// TIA Portal V17 export
// export: Created 2024-06-14T09:53:00.9899822Z, ExportSetting WithDefaults, DisplayName Totally Integrated Automation Portal, DisplayVersion V17, DisplayName TIA Portal Openness, DisplayVersion V17, DisplayName TIA Portal Version Control Interface, DisplayVersion V17, DisplayName Simotion SCOUT TIA, DisplayVersion 5.4.3.0, DisplayName SINAMICS Startdrive Advanced, DisplayVersion V17 SP1 Update 1, DisplayName SINAMICS Startdrive G110M, G120, G120C, G120D, G120P, G115D, DisplayVersion V17 SP1 Update 1, DisplayName SINAMICS Startdrive G130, G150, S120, S150, SINAMICS MV, S210, DisplayVersion V17 SP1 Update 1, DisplayName STEP 7 Professional, DisplayVersion V17, DisplayName STEP 7 Safety, DisplayVersion V17, DisplayName WinCC Professional, DisplayVersion V17
FUNCTION_BLOCK "keypad_logic"   // FB6, LAD
{ S7_Optimized_Access := 'TRUE' }
VERSION : 0.1
// stored: AutoNumber true, IsIECCheckEnabled false, IsRetainMemResEnabled false, MemoryReserve 100, SetENOAutomatically false, UDAEnableTagReadback false
   VAR_INPUT
      Num_0 : Bool;
      Num_1 : Bool;
      Num_2 : Bool;
      Num_3 : Bool;
      Num_4 : Bool;
      Num_5 : Bool;
      Num_6 : Bool;
      Num_7 : Bool;
      Num_8 : Bool;
      Num_9 : Bool;
      enter : Bool;
      clear : Bool;
   END_VAR
   VAR
      count_0 : CTU_INT;
   END_VAR
   VAR RETAIN
      Tens { S7_SetPoint := 'True'} : Int;
   END_VAR
   VAR
      ones : Int;
      decimal : Int;
      P_TRIG : Bool;
      MUL : Int;
      MUL_1 : Int;
      Tare_weight : Real;
      "count _reset" : Bool;
      Tare_Entry : Real;
      "screen count" : Int;
      screen_number : Int;
      screen_reset : Bool;
      MUL_2 : Int;
      count_1 : CTU_INT;
      count_cv_1 : Int;
      "BPCL COUNT" : Int;
      DOMESTIC : Bool;
      COMMERCIAL : Bool;
      MALALBAR_COUNT : Int;
   END_VAR
   VAR RETAIN
      SENSE_1 : Int;
      SENSE_2 : Int;
      SENSE_3 : Int;
      SENSE_4 : Int;
   END_VAR
   VAR
      "SENSI NG_TIME" : Int;
      sens_reset : Bool;
      "open screen" : Bool;
      DOMESTIC_1 : Bool;
      COMMERCIAL_1 : Bool;
      count_2 : CTU_INT;
   END_VAR
   VAR RETAIN
      password { S7_SetPoint := 'True'} : Int;
   END_VAR
   VAR
      password_1 : Int;
      password_2 : Int;
      password_3 : Int;
      password_4 : Int;
      password_5 : Int;
      mul_3 : Int;
      mul_4 : Int;
      mul_5 : Int;
      mul_6 : Int;
      password_reset : Bool;
      sens : Bool;
   END_VAR
   VAR_TEMP
      value_0 : Int;
      count_cv_0 : Int;
   END_VAR
   VAR_TEMP   // added for the SCL form of the ladder/FBD networks
      _w1 : Bool;
      _w2 : Bool;
      _w3 : Bool;
      _w4 : Bool;
      _w5 : Bool;
      _w6 : Bool;
   END_VAR
BEGIN

REGION Network 1
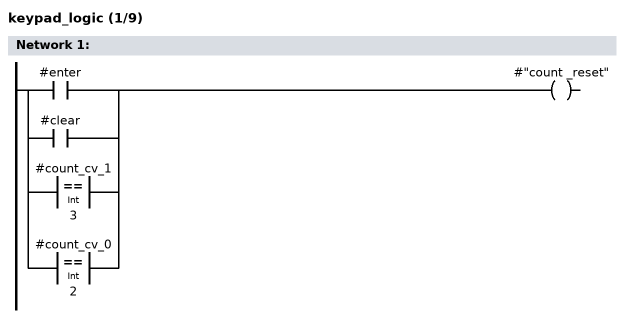
   RUNG wire#powerrail
      Contact( #enter )
      wire#w1
      Coil( #"count _reset" )
   END_RUNG
   RUNG wire#powerrail
      Contact( #clear )
   END_RUNG wire#w1
   RUNG wire#powerrail
      { S7_Templates := "SrcType := Int" } EQ_Contact(in1 := #count_cv_1, in2 := 3)
   END_RUNG wire#w1
   RUNG wire#powerrail
      { S7_Templates := "SrcType := Int" } EQ_Contact(in1 := #count_cv_0, in2 := 2)
   END_RUNG wire#w1
   // the same network as SCL:
   #"count _reset" := #enter OR #clear OR (#count_cv_1 = 3) OR (#count_cv_0 = 2);
END_REGION

REGION Network 2
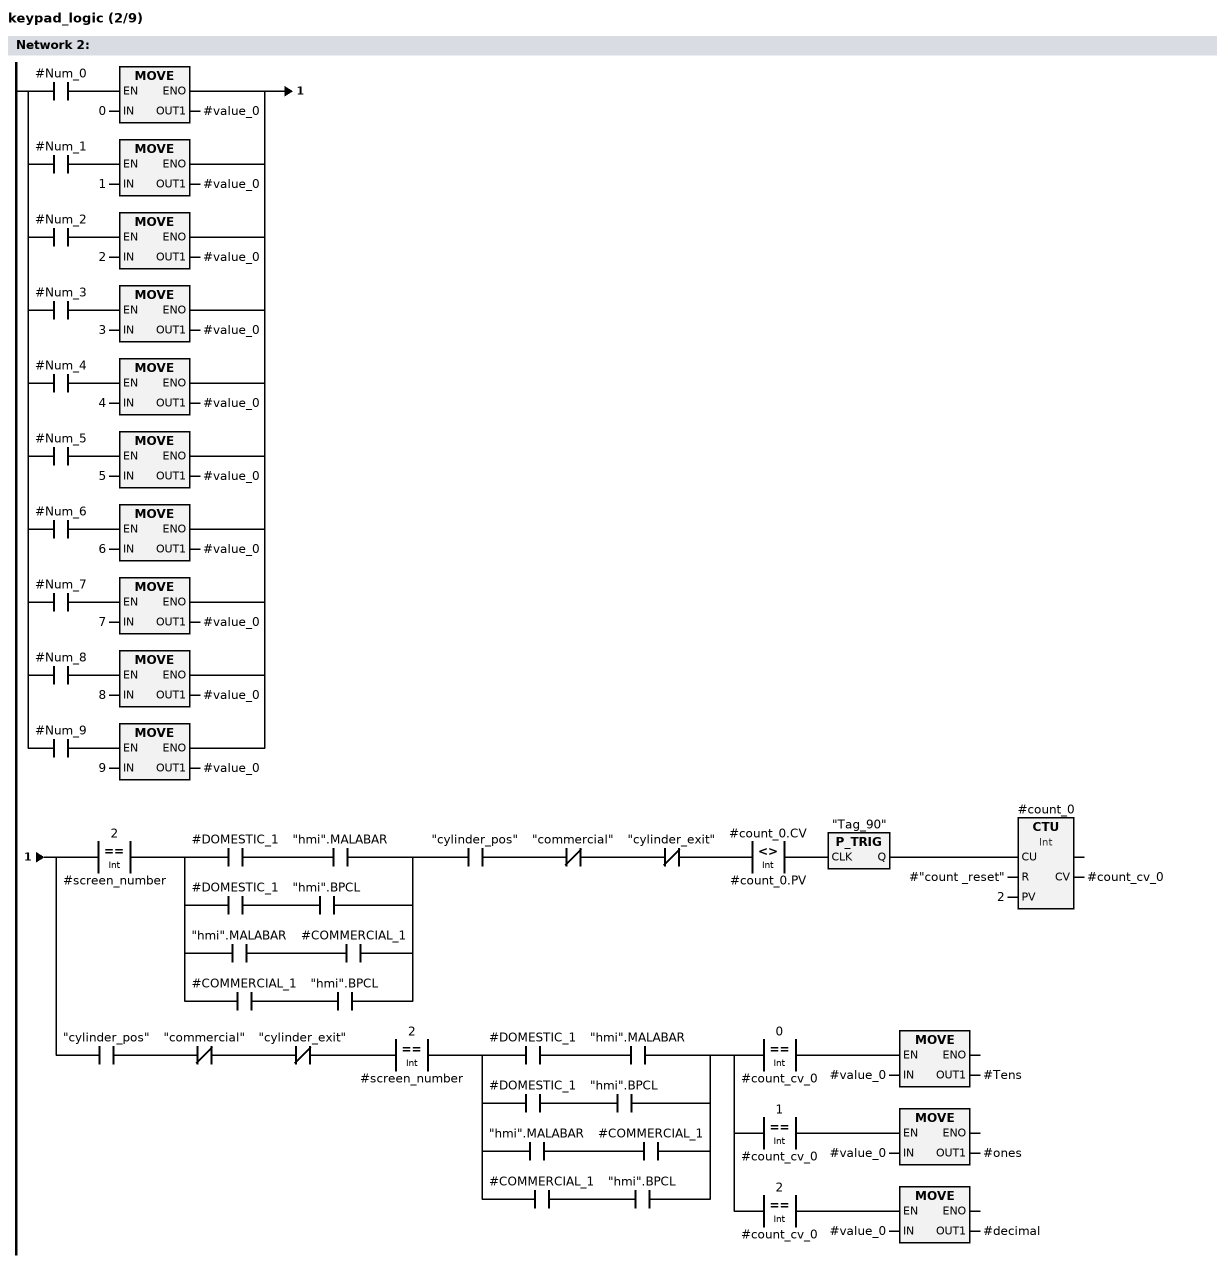
   RUNG wire#powerrail
      Contact( #Num_0 )
      Move(in := 0, out1 => #value_0)
      wire#w1
      { S7_Templates := "SrcType := Int" } EQ_Contact(in1 := 2, in2 := #screen_number)
      wire#w2
      Contact( #DOMESTIC_1 )
      Contact( "hmi".MALABAR )
      wire#w3
      Contact( "cylinder_pos" )
      I_Contact( "commercial" )
      I_Contact( "cylinder_exit" )
      { S7_Templates := "SrcType := Int" } NE_Contact(in1 := #count_0.CV, in2 := #count_0.PV)
      P_Trig( "Tag_90" )
      { S7_Templates := "value_type := Int" } #count_0.CTU(r := #"count _reset", pv := 2, cv => #count_cv_0)
   END_RUNG
   RUNG wire#powerrail
      Contact( #Num_1 )
      Move(in := 1, out1 => #value_0)
   END_RUNG wire#w1
   RUNG wire#powerrail
      Contact( #Num_2 )
      Move(in := 2, out1 => #value_0)
   END_RUNG wire#w1
   RUNG wire#powerrail
      Contact( #Num_3 )
      Move(in := 3, out1 => #value_0)
   END_RUNG wire#w1
   RUNG wire#powerrail
      Contact( #Num_4 )
      Move(in := 4, out1 => #value_0)
   END_RUNG wire#w1
   RUNG wire#powerrail
      Contact( #Num_5 )
      Move(in := 5, out1 => #value_0)
   END_RUNG wire#w1
   RUNG wire#powerrail
      Contact( #Num_6 )
      Move(in := 6, out1 => #value_0)
   END_RUNG wire#w1
   RUNG wire#powerrail
      Contact( #Num_7 )
      Move(in := 7, out1 => #value_0)
   END_RUNG wire#w1
   RUNG wire#powerrail
      Contact( #Num_8 )
      Move(in := 8, out1 => #value_0)
   END_RUNG wire#w1
   RUNG wire#powerrail
      Contact( #Num_9 )
      Move(in := 9, out1 => #value_0)
   END_RUNG wire#w1
   RUNG wire#w2
      Contact( #DOMESTIC_1 )
      Contact( "hmi".BPCL )
   END_RUNG wire#w3
   RUNG wire#w2
      Contact( "hmi".MALABAR )
      Contact( #COMMERCIAL_1 )
   END_RUNG wire#w3
   RUNG wire#w2
      Contact( #COMMERCIAL_1 )
      Contact( "hmi".BPCL )
   END_RUNG wire#w3
   RUNG wire#w1
      Contact( "cylinder_pos" )
      I_Contact( "commercial" )
      I_Contact( "cylinder_exit" )
      { S7_Templates := "SrcType := Int" } EQ_Contact(in1 := 2, in2 := #screen_number)
      wire#w4
      Contact( #DOMESTIC_1 )
      Contact( "hmi".MALABAR )
      wire#w5
      { S7_Templates := "SrcType := Int" } EQ_Contact(in1 := 0, in2 := #count_cv_0)
      Move(in := #value_0, out1 => #Tens)
   END_RUNG
   RUNG wire#w4
      Contact( #DOMESTIC_1 )
      Contact( "hmi".BPCL )
   END_RUNG wire#w5
   RUNG wire#w4
      Contact( "hmi".MALABAR )
      Contact( #COMMERCIAL_1 )
   END_RUNG wire#w5
   RUNG wire#w4
      Contact( #COMMERCIAL_1 )
      Contact( "hmi".BPCL )
   END_RUNG wire#w5
   RUNG wire#w5
      { S7_Templates := "SrcType := Int" } EQ_Contact(in1 := 1, in2 := #count_cv_0)
      Move(in := #value_0, out1 => #ones)
   END_RUNG
   RUNG wire#w5
      { S7_Templates := "SrcType := Int" } EQ_Contact(in1 := 2, in2 := #count_cv_0)
      Move(in := #value_0, out1 => #decimal)
   END_RUNG
   // the same network as SCL:
   IF #Num_0 THEN #value_0 := 0; END_IF;
   IF #Num_1 THEN #value_0 := 1; END_IF;
   IF #Num_2 THEN #value_0 := 2; END_IF;
   IF #Num_3 THEN #value_0 := 3; END_IF;
   IF #Num_4 THEN #value_0 := 4; END_IF;
   IF #Num_5 THEN #value_0 := 5; END_IF;
   IF #Num_6 THEN #value_0 := 6; END_IF;
   IF #Num_7 THEN #value_0 := 7; END_IF;
   IF #Num_8 THEN #value_0 := 8; END_IF;
   IF #Num_9 THEN #value_0 := 9; END_IF;
   #_w1 := #Num_0 OR #Num_1 OR #Num_2 OR #Num_3 OR #Num_4 OR #Num_5 OR #Num_6 OR #Num_7 OR #Num_8 OR #Num_9;
   #_w2 := #_w1 AND (2 = #screen_number) AND ((#DOMESTIC_1 AND "hmi".MALABAR) OR (#DOMESTIC_1 AND "hmi".BPCL) OR ("hmi".MALABAR AND #COMMERCIAL_1) OR (#COMMERCIAL_1 AND "hmi".BPCL)) AND "cylinder_pos" AND NOT "commercial" AND NOT "cylinder_exit" AND (#count_0.CV <> #count_0.PV);
   #_w3 := #_w2 AND NOT "Tag_90";   // rising edge
   "Tag_90" := #_w2;
   #count_0(CU := #_w3, R := #"count _reset", PV := 2, CV => #count_cv_0);   // CTU
   #_w4 := #_w1 AND "cylinder_pos" AND NOT "commercial" AND NOT "cylinder_exit" AND (2 = #screen_number) AND ((#DOMESTIC_1 AND "hmi".MALABAR) OR (#DOMESTIC_1 AND "hmi".BPCL) OR ("hmi".MALABAR AND #COMMERCIAL_1) OR (#COMMERCIAL_1 AND "hmi".BPCL));
   IF #_w4 AND (0 = #count_cv_0) THEN #Tens := #value_0; END_IF;
   IF #_w4 AND (1 = #count_cv_0) THEN #ones := #value_0; END_IF;
   IF #_w4 AND (2 = #count_cv_0) THEN #decimal := #value_0; END_IF;
END_REGION

REGION Network 3
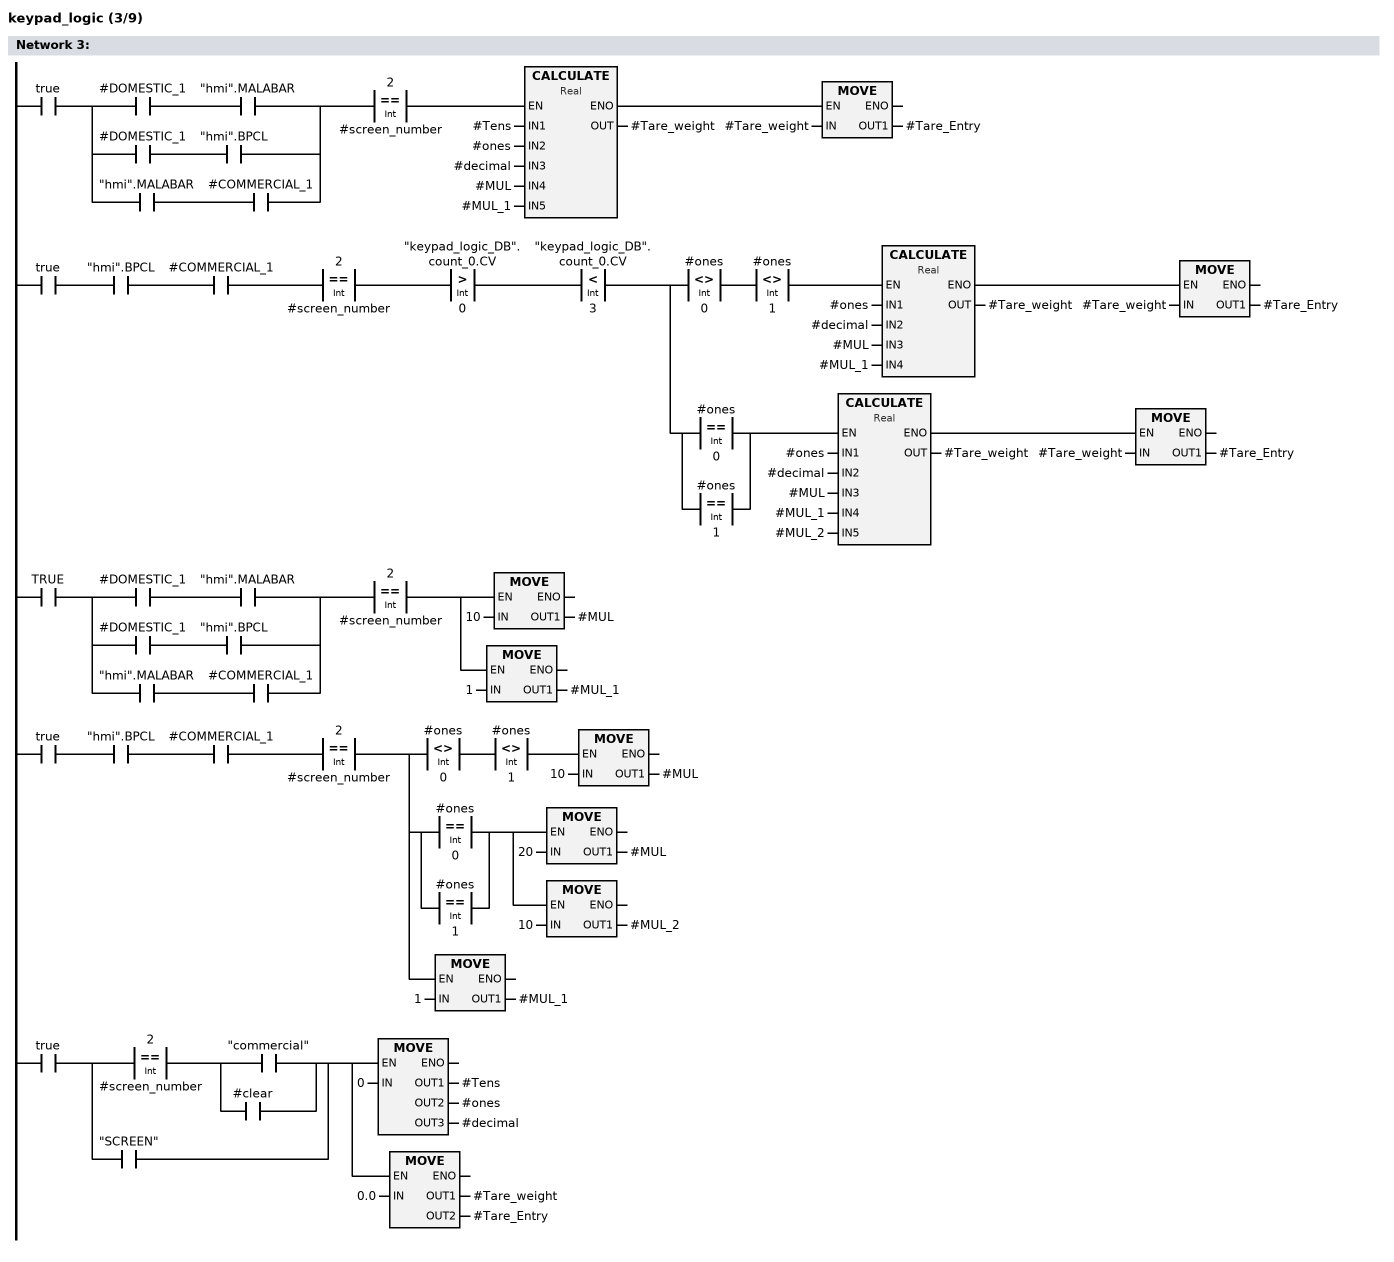
   RUNG wire#powerrail
      Contact( true )
      wire#w1
      Contact( #DOMESTIC_1 )
      Contact( "hmi".MALABAR )
      wire#w2
      { S7_Templates := "SrcType := Int" } EQ_Contact(in1 := 2, in2 := #screen_number)
      { S7_Templates := "SrcType := Real"; S7_Expression := "IN4+(IN2*IN5)+(IN3/IN4)" } Calculate(in1 := #Tens, in2 := #ones, in3 := #decimal, in4 := #MUL, in5 := #MUL_1, out => #Tare_weight)
      Move(in := #Tare_weight, out1 => #Tare_Entry)
   END_RUNG
   RUNG wire#w1
      Contact( #DOMESTIC_1 )
      Contact( "hmi".BPCL )
   END_RUNG wire#w2
   RUNG wire#w1
      Contact( "hmi".MALABAR )
      Contact( #COMMERCIAL_1 )
   END_RUNG wire#w2
   RUNG wire#powerrail
      Contact( true )
      Contact( "hmi".BPCL )
      Contact( #COMMERCIAL_1 )
      { S7_Templates := "SrcType := Int" } EQ_Contact(in1 := 2, in2 := #screen_number)
      { S7_Templates := "SrcType := Int" } GT_Contact(in1 := "keypad_logic_DB".count_0.CV, in2 := 0)
      { S7_Templates := "SrcType := Int" } LT_Contact(in1 := "keypad_logic_DB".count_0.CV, in2 := 3)
      wire#w3
      { S7_Templates := "SrcType := Int" } NE_Contact(in1 := #ones, in2 := 0)
      { S7_Templates := "SrcType := Int" } NE_Contact(in1 := #ones, in2 := 1)
      { S7_Templates := "SrcType := Real"; S7_Expression := "IN3+(IN1*IN4)+(IN2/IN3)" } Calculate(in1 := #ones, in2 := #decimal, in3 := #MUL, in4 := #MUL_1, out => #Tare_weight)
      Move(in := #Tare_weight, out1 => #Tare_Entry)
   END_RUNG
   RUNG wire#w3
      { S7_Templates := "SrcType := Int" } EQ_Contact(in1 := #ones, in2 := 0)
      wire#w4
      { S7_Templates := "SrcType := Real"; S7_Expression := "IN3+(IN1*IN4)+(IN2/IN5)" } Calculate(in1 := #ones, in2 := #decimal, in3 := #MUL, in4 := #MUL_1, in5 := #MUL_2, out => #Tare_weight)
      Move(in := #Tare_weight, out1 => #Tare_Entry)
   END_RUNG
   RUNG wire#w3
      { S7_Templates := "SrcType := Int" } EQ_Contact(in1 := #ones, in2 := 1)
   END_RUNG wire#w4
   RUNG wire#powerrail
      Contact( TRUE )
      wire#w5
      Contact( #DOMESTIC_1 )
      Contact( "hmi".MALABAR )
      wire#w6
      { S7_Templates := "SrcType := Int" } EQ_Contact(in1 := 2, in2 := #screen_number)
      wire#w7
      Move(in := 10, out1 => #MUL)
   END_RUNG
   RUNG wire#w5
      Contact( #DOMESTIC_1 )
      Contact( "hmi".BPCL )
   END_RUNG wire#w6
   RUNG wire#w5
      Contact( "hmi".MALABAR )
      Contact( #COMMERCIAL_1 )
   END_RUNG wire#w6
   RUNG wire#w7
      Move(in := 1, out1 => #MUL_1)
   END_RUNG
   RUNG wire#powerrail
      Contact( true )
      Contact( "hmi".BPCL )
      Contact( #COMMERCIAL_1 )
      { S7_Templates := "SrcType := Int" } EQ_Contact(in1 := 2, in2 := #screen_number)
      wire#w8
      { S7_Templates := "SrcType := Int" } NE_Contact(in1 := #ones, in2 := 0)
      { S7_Templates := "SrcType := Int" } NE_Contact(in1 := #ones, in2 := 1)
      Move(in := 10, out1 => #MUL)
   END_RUNG
   RUNG wire#w8
      { S7_Templates := "SrcType := Int" } EQ_Contact(in1 := #ones, in2 := 0)
      wire#w9
      Move(in := 20, out1 => #MUL)
   END_RUNG
   RUNG wire#w8
      { S7_Templates := "SrcType := Int" } EQ_Contact(in1 := #ones, in2 := 1)
   END_RUNG wire#w9
   RUNG wire#w9
      Move(in := 10, out1 => #MUL_2)
   END_RUNG
   RUNG wire#w8
      Move(in := 1, out1 => #MUL_1)
   END_RUNG
   RUNG wire#powerrail
      Contact( true )
      wire#w10
      { S7_Templates := "SrcType := Int" } EQ_Contact(in1 := 2, in2 := #screen_number)
      wire#w11
      Contact( "commercial" )
      wire#w12
      Move(in := 0, out1 => #Tens, out2 => #ones, out3 => #decimal)
   END_RUNG
   RUNG wire#w11
      Contact( #clear )
   END_RUNG wire#w12
   RUNG wire#w10
      Contact( "SCREEN" )
   END_RUNG wire#w12
   RUNG wire#w12
      Move(in := 0.0, out1 => #Tare_weight, out2 => #Tare_Entry)
   END_RUNG
   // the same network as SCL:
   IF true AND ((#DOMESTIC_1 AND "hmi".MALABAR) OR (#DOMESTIC_1 AND "hmi".BPCL) OR ("hmi".MALABAR AND #COMMERCIAL_1)) AND (2 = #screen_number) THEN
       #Tare_weight := #MUL+(#ones*#MUL_1)+(#decimal/#MUL);
       #Tare_Entry := #Tare_weight;
   END_IF;
   #_w1 := true AND "hmi".BPCL AND #COMMERCIAL_1 AND (2 = #screen_number) AND ("keypad_logic_DB".count_0.CV > 0) AND ("keypad_logic_DB".count_0.CV < 3);
   IF #_w1 AND (#ones <> 0) AND (#ones <> 1) THEN
       #Tare_weight := #MUL+(#ones*#MUL_1)+(#decimal/#MUL);
       #Tare_Entry := #Tare_weight;
   END_IF;
   IF #_w1 AND ((#ones = 0) OR (#ones = 1)) THEN
       #Tare_weight := #MUL+(#ones*#MUL_1)+(#decimal/#MUL_2);
       #Tare_Entry := #Tare_weight;
   END_IF;
   IF TRUE AND ((#DOMESTIC_1 AND "hmi".MALABAR) OR (#DOMESTIC_1 AND "hmi".BPCL) OR ("hmi".MALABAR AND #COMMERCIAL_1)) AND (2 = #screen_number) THEN
       #MUL := 10;
       #MUL_1 := 1;
   END_IF;
   #_w2 := true AND "hmi".BPCL AND #COMMERCIAL_1 AND (2 = #screen_number);
   IF #_w2 AND (#ones <> 0) AND (#ones <> 1) THEN #MUL := 10; END_IF;
   IF #_w2 AND ((#ones = 0) OR (#ones = 1)) THEN
       #MUL := 20;
       #MUL_2 := 10;
   END_IF;
   IF #_w2 THEN #MUL_1 := 1; END_IF;
   IF true AND (((2 = #screen_number) AND ("commercial" OR #clear)) OR "SCREEN") THEN
       #Tens := 0;
       #ones := 0;
       #decimal := 0;
       #Tare_weight := 0.0;
       #Tare_Entry := 0.0;
   END_IF;
END_REGION

REGION Network 4
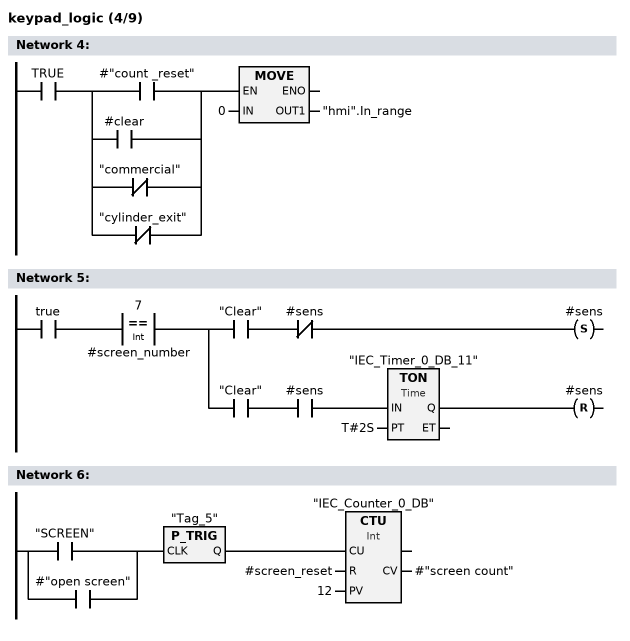
   RUNG wire#powerrail
      Contact( TRUE )
      wire#w1
      Contact( #"count _reset" )
      wire#w2
      Move(in := 0, out1 => "hmi".In_range)
   END_RUNG
   RUNG wire#w1
      Contact( #clear )
   END_RUNG wire#w2
   RUNG wire#w1
      I_Contact( "commercial" )
   END_RUNG wire#w2
   RUNG wire#w1
      I_Contact( "cylinder_exit" )
   END_RUNG wire#w2
   // the same network as SCL:
   IF TRUE AND (#"count _reset" OR #clear OR NOT "commercial" OR NOT "cylinder_exit") THEN
       "hmi".In_range := 0;
   END_IF;
END_REGION

REGION Network 5
   RUNG wire#powerrail
      Contact( true )
      { S7_Templates := "SrcType := Int" } EQ_Contact(in1 := 7, in2 := #screen_number)
      wire#w1
      Contact( "Clear" )
      I_Contact( #sens )
      S_Coil( #sens )
   END_RUNG
   RUNG wire#w1
      Contact( "Clear" )
      Contact( #sens )
      { S7_Templates := "time_type := Time" } "IEC_Timer_0_DB_11".TON(pt := T#2S, et =>)
      R_Coil( #sens )
   END_RUNG
   // the same network as SCL:
   #_w1 := true AND (7 = #screen_number);
   IF #_w1 AND "Clear" AND NOT #sens THEN #sens := TRUE; END_IF;
   "IEC_Timer_0_DB_11".TON(IN := #_w1 AND "Clear" AND #sens, PT := T#2S);
   IF "IEC_Timer_0_DB_11".Q THEN #sens := FALSE; END_IF;
END_REGION

REGION Network 6
   RUNG wire#powerrail
      Contact( "SCREEN" )
      wire#w1
      P_Trig( "Tag_5" )
      { S7_Templates := "value_type := Int" } "IEC_Counter_0_DB".CTU(r := #screen_reset, pv := 12, cv => #"screen count")
   END_RUNG
   RUNG wire#powerrail
      Contact( #"open screen" )
   END_RUNG wire#w1
   // the same network as SCL:
   #_w1 := "SCREEN" OR #"open screen";
   #_w2 := #_w1 AND NOT "Tag_5";   // rising edge
   "Tag_5" := #_w1;
   "IEC_Counter_0_DB".CTU(CU := #_w2, R := #screen_reset, PV := 12, CV => #"screen count");
END_REGION

REGION Network 7
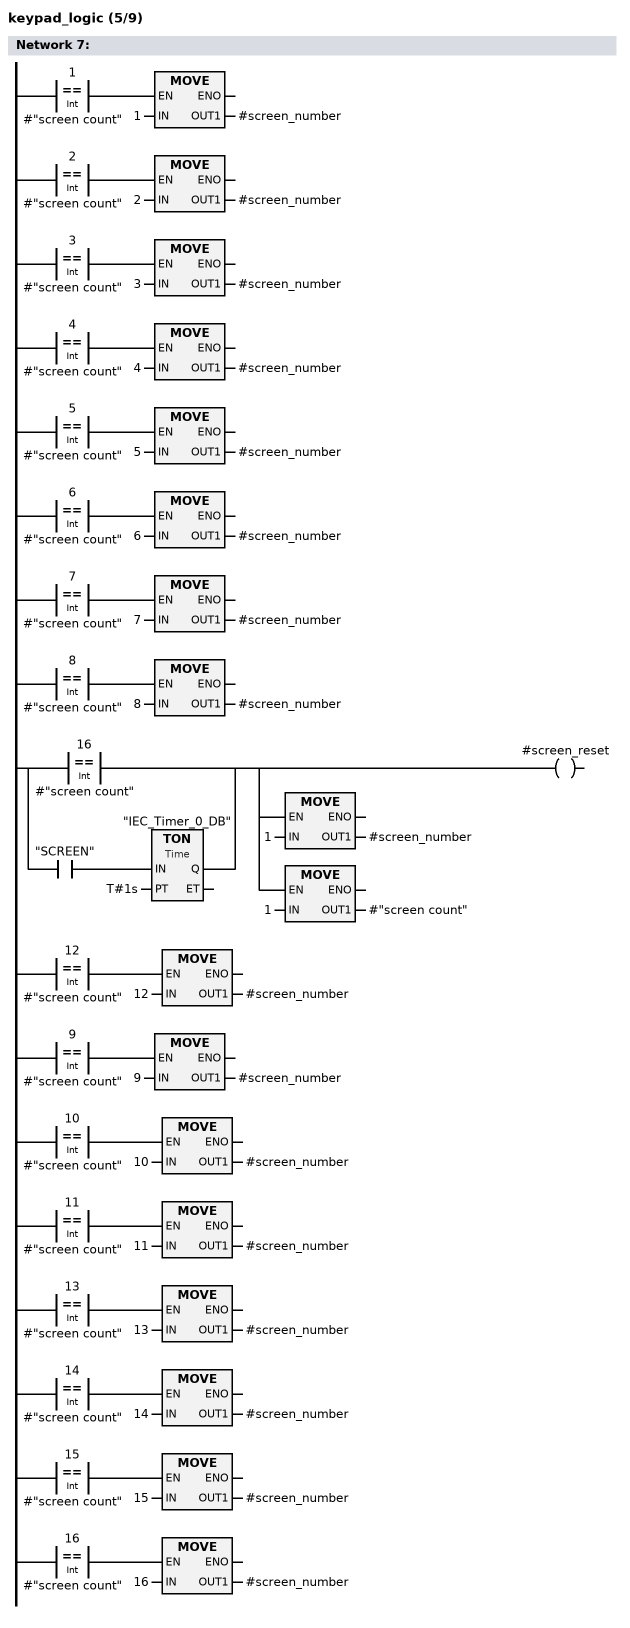
   RUNG wire#powerrail
      { S7_Templates := "SrcType := Int" } EQ_Contact(in1 := 1, in2 := #"screen count")
      Move(in := 1, out1 => #screen_number)
   END_RUNG
   RUNG wire#powerrail
      { S7_Templates := "SrcType := Int" } EQ_Contact(in1 := 2, in2 := #"screen count")
      Move(in := 2, out1 => #screen_number)
   END_RUNG
   RUNG wire#powerrail
      { S7_Templates := "SrcType := Int" } EQ_Contact(in1 := 3, in2 := #"screen count")
      Move(in := 3, out1 => #screen_number)
   END_RUNG
   RUNG wire#powerrail
      { S7_Templates := "SrcType := Int" } EQ_Contact(in1 := 4, in2 := #"screen count")
      Move(in := 4, out1 => #screen_number)
   END_RUNG
   RUNG wire#powerrail
      { S7_Templates := "SrcType := Int" } EQ_Contact(in1 := 5, in2 := #"screen count")
      Move(in := 5, out1 => #screen_number)
   END_RUNG
   RUNG wire#powerrail
      { S7_Templates := "SrcType := Int" } EQ_Contact(in1 := 6, in2 := #"screen count")
      Move(in := 6, out1 => #screen_number)
   END_RUNG
   RUNG wire#powerrail
      { S7_Templates := "SrcType := Int" } EQ_Contact(in1 := 7, in2 := #"screen count")
      Move(in := 7, out1 => #screen_number)
   END_RUNG
   RUNG wire#powerrail
      { S7_Templates := "SrcType := Int" } EQ_Contact(in1 := 8, in2 := #"screen count")
      Move(in := 8, out1 => #screen_number)
   END_RUNG
   RUNG wire#powerrail
      { S7_Templates := "SrcType := Int" } EQ_Contact(in1 := 16, in2 := #"screen count")
      wire#w1
      Coil( #screen_reset )
   END_RUNG
   RUNG wire#powerrail
      Contact( "SCREEN" )
      { S7_Templates := "time_type := Time" } "IEC_Timer_0_DB".TON(pt := T#1s, et =>)
   END_RUNG wire#w1
   RUNG wire#w1
      Move(in := 1, out1 => #screen_number)
   END_RUNG
   RUNG wire#w1
      Move(in := 1, out1 => #"screen count")
   END_RUNG
   RUNG wire#powerrail
      { S7_Templates := "SrcType := Int" } EQ_Contact(in1 := 12, in2 := #"screen count")
      Move(in := 12, out1 => #screen_number)
   END_RUNG
   RUNG wire#powerrail
      { S7_Templates := "SrcType := Int" } EQ_Contact(in1 := 9, in2 := #"screen count")
      Move(in := 9, out1 => #screen_number)
   END_RUNG
   RUNG wire#powerrail
      { S7_Templates := "SrcType := Int" } EQ_Contact(in1 := 10, in2 := #"screen count")
      Move(in := 10, out1 => #screen_number)
   END_RUNG
   RUNG wire#powerrail
      { S7_Templates := "SrcType := Int" } EQ_Contact(in1 := 11, in2 := #"screen count")
      Move(in := 11, out1 => #screen_number)
   END_RUNG
   RUNG wire#powerrail
      { S7_Templates := "SrcType := Int" } EQ_Contact(in1 := 13, in2 := #"screen count")
      Move(in := 13, out1 => #screen_number)
   END_RUNG
   RUNG wire#powerrail
      { S7_Templates := "SrcType := Int" } EQ_Contact(in1 := 14, in2 := #"screen count")
      Move(in := 14, out1 => #screen_number)
   END_RUNG
   RUNG wire#powerrail
      { S7_Templates := "SrcType := Int" } EQ_Contact(in1 := 15, in2 := #"screen count")
      Move(in := 15, out1 => #screen_number)
   END_RUNG
   RUNG wire#powerrail
      { S7_Templates := "SrcType := Int" } EQ_Contact(in1 := 16, in2 := #"screen count")
      Move(in := 16, out1 => #screen_number)
   END_RUNG
   // the same network as SCL:
   IF 1 = #"screen count" THEN #screen_number := 1; END_IF;
   IF 2 = #"screen count" THEN #screen_number := 2; END_IF;
   IF 3 = #"screen count" THEN #screen_number := 3; END_IF;
   IF 4 = #"screen count" THEN #screen_number := 4; END_IF;
   IF 5 = #"screen count" THEN #screen_number := 5; END_IF;
   IF 6 = #"screen count" THEN #screen_number := 6; END_IF;
   IF 7 = #"screen count" THEN #screen_number := 7; END_IF;
   IF 8 = #"screen count" THEN #screen_number := 8; END_IF;
   "IEC_Timer_0_DB".TON(IN := "SCREEN", PT := T#1s);
   #screen_reset := (16 = #"screen count") OR "IEC_Timer_0_DB".Q;
   IF #screen_reset THEN
       #screen_number := 1;
       #"screen count" := 1;
   END_IF;
   IF 12 = #"screen count" THEN #screen_number := 12; END_IF;
   IF 9 = #"screen count" THEN #screen_number := 9; END_IF;
   IF 10 = #"screen count" THEN #screen_number := 10; END_IF;
   IF 11 = #"screen count" THEN #screen_number := 11; END_IF;
   IF 13 = #"screen count" THEN #screen_number := 13; END_IF;
   IF 14 = #"screen count" THEN #screen_number := 14; END_IF;
   IF 15 = #"screen count" THEN #screen_number := 15; END_IF;
   IF 16 = #"screen count" THEN #screen_number := 16; END_IF;
END_REGION

REGION Network 8
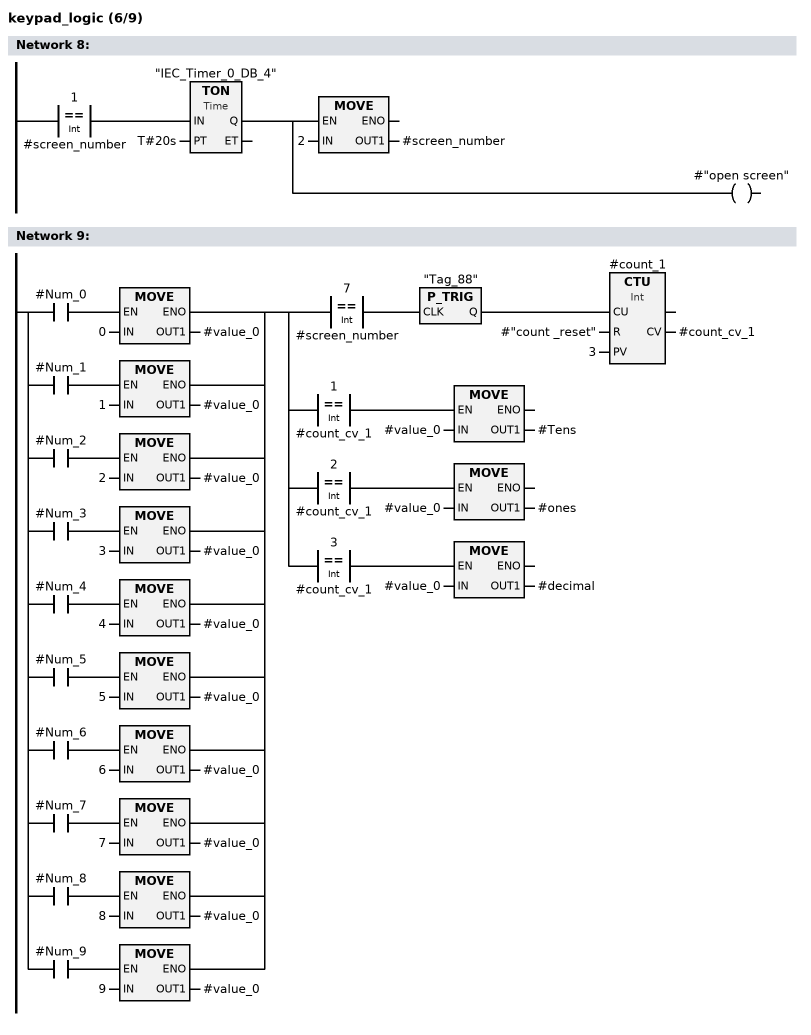
   RUNG wire#powerrail
      { S7_Templates := "SrcType := Int" } EQ_Contact(in1 := 1, in2 := #screen_number)
      { S7_Templates := "time_type := Time" } "IEC_Timer_0_DB_4".TON(pt := T#20s, et =>)
      wire#w1
      Move(in := 2, out1 => #screen_number)
   END_RUNG
   RUNG wire#w1
      Coil( #"open screen" )
   END_RUNG
   // the same network as SCL:
   "IEC_Timer_0_DB_4".TON(IN := 1 = #screen_number, PT := T#20s);
   IF "IEC_Timer_0_DB_4".Q THEN #screen_number := 2; END_IF;
   #"open screen" := "IEC_Timer_0_DB_4".Q;
END_REGION

REGION Network 9
   RUNG wire#powerrail
      Contact( #Num_0 )
      Move(in := 0, out1 => #value_0)
      wire#w1
      { S7_Templates := "SrcType := Int" } EQ_Contact(in1 := 7, in2 := #screen_number)
      P_Trig( "Tag_88" )
      { S7_Templates := "value_type := Int" } #count_1.CTU(r := #"count _reset", pv := 3, cv => #count_cv_1)
   END_RUNG
   RUNG wire#powerrail
      Contact( #Num_1 )
      Move(in := 1, out1 => #value_0)
   END_RUNG wire#w1
   RUNG wire#powerrail
      Contact( #Num_2 )
      Move(in := 2, out1 => #value_0)
   END_RUNG wire#w1
   RUNG wire#powerrail
      Contact( #Num_3 )
      Move(in := 3, out1 => #value_0)
   END_RUNG wire#w1
   RUNG wire#powerrail
      Contact( #Num_4 )
      Move(in := 4, out1 => #value_0)
   END_RUNG wire#w1
   RUNG wire#powerrail
      Contact( #Num_5 )
      Move(in := 5, out1 => #value_0)
   END_RUNG wire#w1
   RUNG wire#powerrail
      Contact( #Num_6 )
      Move(in := 6, out1 => #value_0)
   END_RUNG wire#w1
   RUNG wire#powerrail
      Contact( #Num_7 )
      Move(in := 7, out1 => #value_0)
   END_RUNG wire#w1
   RUNG wire#powerrail
      Contact( #Num_8 )
      Move(in := 8, out1 => #value_0)
   END_RUNG wire#w1
   RUNG wire#powerrail
      Contact( #Num_9 )
      Move(in := 9, out1 => #value_0)
   END_RUNG wire#w1
   RUNG wire#w1
      { S7_Templates := "SrcType := Int" } EQ_Contact(in1 := 1, in2 := #count_cv_1)
      Move(in := #value_0, out1 => #Tens)
   END_RUNG
   RUNG wire#w1
      { S7_Templates := "SrcType := Int" } EQ_Contact(in1 := 2, in2 := #count_cv_1)
      Move(in := #value_0, out1 => #ones)
   END_RUNG
   RUNG wire#w1
      { S7_Templates := "SrcType := Int" } EQ_Contact(in1 := 3, in2 := #count_cv_1)
      Move(in := #value_0, out1 => #decimal)
   END_RUNG
   // the same network as SCL:
   IF #Num_0 THEN #value_0 := 0; END_IF;
   IF #Num_1 THEN #value_0 := 1; END_IF;
   IF #Num_2 THEN #value_0 := 2; END_IF;
   IF #Num_3 THEN #value_0 := 3; END_IF;
   IF #Num_4 THEN #value_0 := 4; END_IF;
   IF #Num_5 THEN #value_0 := 5; END_IF;
   IF #Num_6 THEN #value_0 := 6; END_IF;
   IF #Num_7 THEN #value_0 := 7; END_IF;
   IF #Num_8 THEN #value_0 := 8; END_IF;
   IF #Num_9 THEN #value_0 := 9; END_IF;
   #_w1 := #Num_0 OR #Num_1 OR #Num_2 OR #Num_3 OR #Num_4 OR #Num_5 OR #Num_6 OR #Num_7 OR #Num_8 OR #Num_9;
   #_w2 := #_w1 AND (7 = #screen_number);
   #_w3 := #_w2 AND NOT "Tag_88";   // rising edge
   "Tag_88" := #_w2;
   #count_1(CU := #_w3, R := #"count _reset", PV := 3, CV => #count_cv_1);   // CTU
   IF #_w1 AND (1 = #count_cv_1) THEN #Tens := #value_0; END_IF;
   IF #_w1 AND (2 = #count_cv_1) THEN #ones := #value_0; END_IF;
   IF #_w1 AND (3 = #count_cv_1) THEN #decimal := #value_0; END_IF;
END_REGION

REGION Network 10
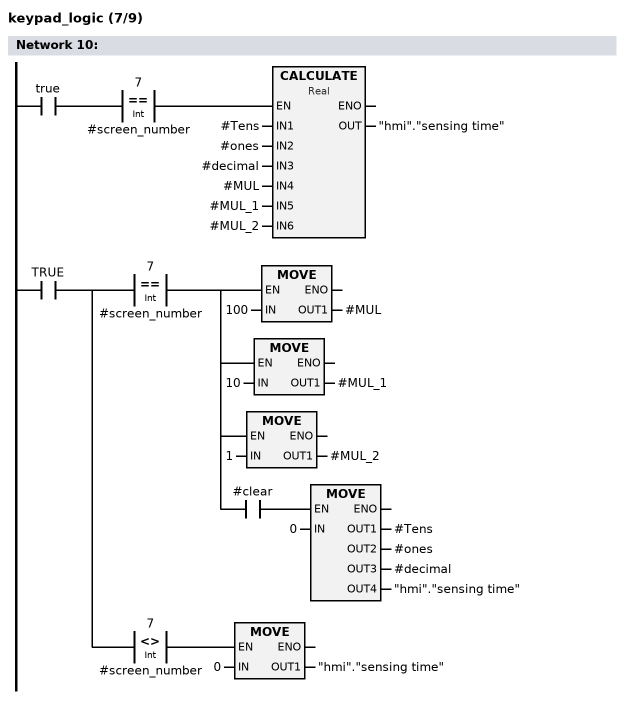
   RUNG wire#powerrail
      Contact( true )
      { S7_Templates := "SrcType := Int" } EQ_Contact(in1 := 7, in2 := #screen_number)
      { S7_Templates := "SrcType := Real"; S7_Expression := "(IN1*IN4)+(IN2*IN5)+(IN3*IN6)" } Calculate(in1 := #Tens, in2 := #ones, in3 := #decimal, in4 := #MUL, in5 := #MUL_1, in6 := #MUL_2, out => "hmi"."sensing time")
   END_RUNG
   RUNG wire#powerrail
      Contact( TRUE )
      wire#w1
      { S7_Templates := "SrcType := Int" } EQ_Contact(in1 := 7, in2 := #screen_number)
      wire#w2
      Move(in := 100, out1 => #MUL)
   END_RUNG
   RUNG wire#w2
      Move(in := 10, out1 => #MUL_1)
   END_RUNG
   RUNG wire#w2
      Move(in := 1, out1 => #MUL_2)
   END_RUNG
   RUNG wire#w2
      Contact( #clear )
      Move(in := 0, out1 => #Tens, out2 => #ones, out3 => #decimal, out4 => "hmi"."sensing time")
   END_RUNG
   RUNG wire#w1
      { S7_Templates := "SrcType := Int" } NE_Contact(in1 := 7, in2 := #screen_number)
      Move(in := 0, out1 => "hmi"."sensing time")
   END_RUNG
   // the same network as SCL:
   IF true AND (7 = #screen_number) THEN
       "hmi"."sensing time" := (#Tens*#MUL)+(#ones*#MUL_1)+(#decimal*#MUL_2);
   END_IF;
   #_w1 := TRUE AND (7 = #screen_number);
   IF #_w1 THEN
       #MUL := 100;
       #MUL_1 := 10;
       #MUL_2 := 1;
   END_IF;
   IF #_w1 AND #clear THEN
       #Tens := 0;
       #ones := 0;
       #decimal := 0;
       "hmi"."sensing time" := 0;
   END_IF;
   IF TRUE AND (7 <> #screen_number) THEN "hmi"."sensing time" := 0; END_IF;
END_REGION

REGION Network 11
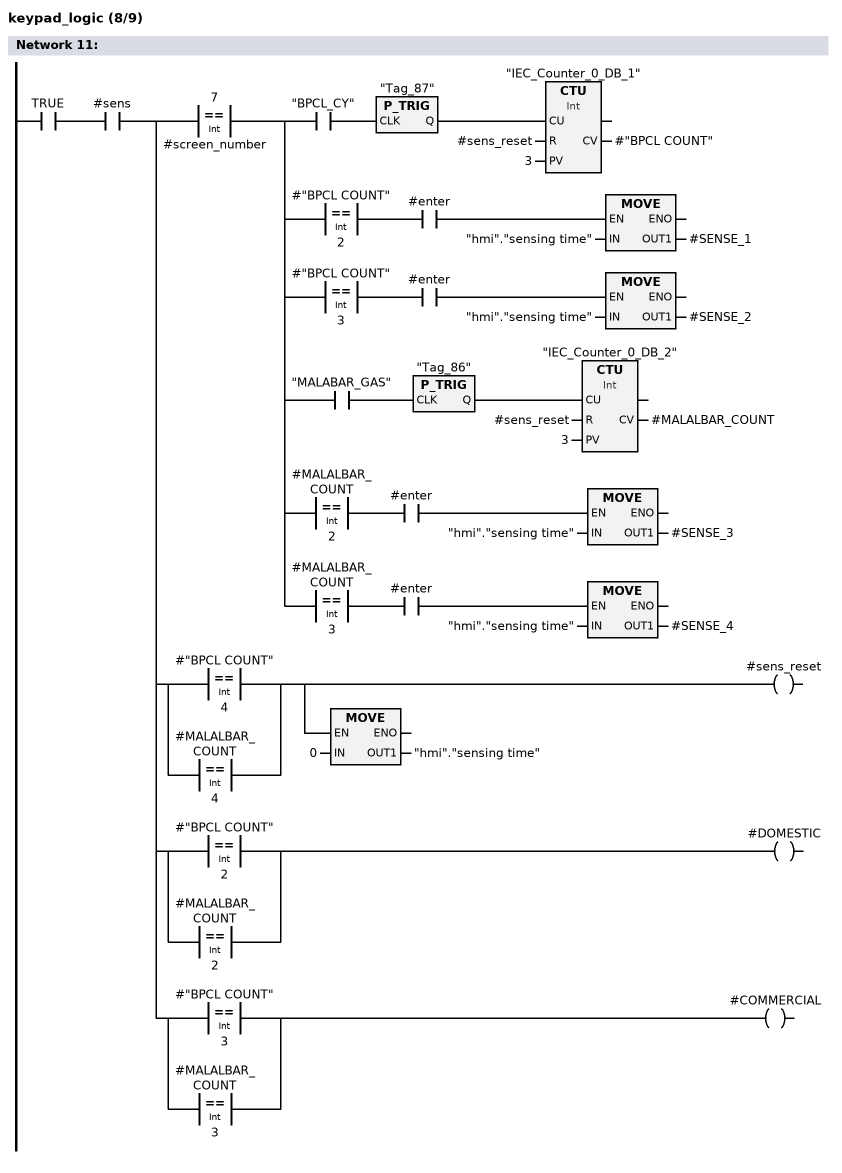
   RUNG wire#powerrail
      Contact( TRUE )
      Contact( #sens )
      wire#w1
      { S7_Templates := "SrcType := Int" } EQ_Contact(in1 := 7, in2 := #screen_number)
      wire#w2
      Contact( "BPCL_CY" )
      P_Trig( "Tag_87" )
      { S7_Templates := "value_type := Int" } "IEC_Counter_0_DB_1".CTU(r := #sens_reset, pv := 3, cv => #"BPCL COUNT")
   END_RUNG
   RUNG wire#w2
      { S7_Templates := "SrcType := Int" } EQ_Contact(in1 := #"BPCL COUNT", in2 := 2)
      Contact( #enter )
      Move(in := "hmi"."sensing time", out1 => #SENSE_1)
   END_RUNG
   RUNG wire#w2
      { S7_Templates := "SrcType := Int" } EQ_Contact(in1 := #"BPCL COUNT", in2 := 3)
      Contact( #enter )
      Move(in := "hmi"."sensing time", out1 => #SENSE_2)
   END_RUNG
   RUNG wire#w2
      Contact( "MALABAR_GAS" )
      P_Trig( "Tag_86" )
      { S7_Templates := "value_type := Int" } "IEC_Counter_0_DB_2".CTU(r := #sens_reset, pv := 3, cv => #MALALBAR_COUNT)
   END_RUNG
   RUNG wire#w2
      { S7_Templates := "SrcType := Int" } EQ_Contact(in1 := #MALALBAR_COUNT, in2 := 2)
      Contact( #enter )
      Move(in := "hmi"."sensing time", out1 => #SENSE_3)
   END_RUNG
   RUNG wire#w2
      { S7_Templates := "SrcType := Int" } EQ_Contact(in1 := #MALALBAR_COUNT, in2 := 3)
      Contact( #enter )
      Move(in := "hmi"."sensing time", out1 => #SENSE_4)
   END_RUNG
   RUNG wire#w1
      { S7_Templates := "SrcType := Int" } EQ_Contact(in1 := #"BPCL COUNT", in2 := 4)
      wire#w3
      Coil( #sens_reset )
   END_RUNG
   RUNG wire#w1
      { S7_Templates := "SrcType := Int" } EQ_Contact(in1 := #MALALBAR_COUNT, in2 := 4)
   END_RUNG wire#w3
   RUNG wire#w3
      Move(in := 0, out1 => "hmi"."sensing time")
   END_RUNG
   RUNG wire#w1
      { S7_Templates := "SrcType := Int" } EQ_Contact(in1 := #"BPCL COUNT", in2 := 2)
      wire#w4
      Coil( #DOMESTIC )
   END_RUNG
   RUNG wire#w1
      { S7_Templates := "SrcType := Int" } EQ_Contact(in1 := #MALALBAR_COUNT, in2 := 2)
   END_RUNG wire#w4
   RUNG wire#w1
      { S7_Templates := "SrcType := Int" } EQ_Contact(in1 := #"BPCL COUNT", in2 := 3)
      wire#w5
      Coil( #COMMERCIAL )
   END_RUNG
   RUNG wire#w1
      { S7_Templates := "SrcType := Int" } EQ_Contact(in1 := #MALALBAR_COUNT, in2 := 3)
   END_RUNG wire#w5
   // the same network as SCL:
   #_w1 := TRUE AND #sens;
   #_w2 := #_w1 AND (7 = #screen_number);
   #_w3 := #_w2 AND "BPCL_CY";
   #_w4 := #_w3 AND NOT "Tag_87";   // rising edge
   "Tag_87" := #_w3;
   "IEC_Counter_0_DB_1".CTU(CU := #_w4, R := #sens_reset, PV := 3, CV => #"BPCL COUNT");
   IF #_w2 AND (#"BPCL COUNT" = 2) AND #enter THEN #SENSE_1 := "hmi"."sensing time"; END_IF;
   IF #_w2 AND (#"BPCL COUNT" = 3) AND #enter THEN #SENSE_2 := "hmi"."sensing time"; END_IF;
   #_w5 := #_w2 AND "MALABAR_GAS";
   #_w6 := #_w5 AND NOT "Tag_86";   // rising edge
   "Tag_86" := #_w5;
   "IEC_Counter_0_DB_2".CTU(CU := #_w6, R := #sens_reset, PV := 3, CV => #MALALBAR_COUNT);
   IF #_w2 AND (#MALALBAR_COUNT = 2) AND #enter THEN #SENSE_3 := "hmi"."sensing time"; END_IF;
   IF #_w2 AND (#MALALBAR_COUNT = 3) AND #enter THEN #SENSE_4 := "hmi"."sensing time"; END_IF;
   #sens_reset := #_w1 AND ((#"BPCL COUNT" = 4) OR (#MALALBAR_COUNT = 4));
   IF #sens_reset THEN "hmi"."sensing time" := 0; END_IF;
   #DOMESTIC := #_w1 AND ((#"BPCL COUNT" = 2) OR (#MALALBAR_COUNT = 2));
   #COMMERCIAL := #_w1 AND ((#"BPCL COUNT" = 3) OR (#MALALBAR_COUNT = 3));
END_REGION

REGION Network 12
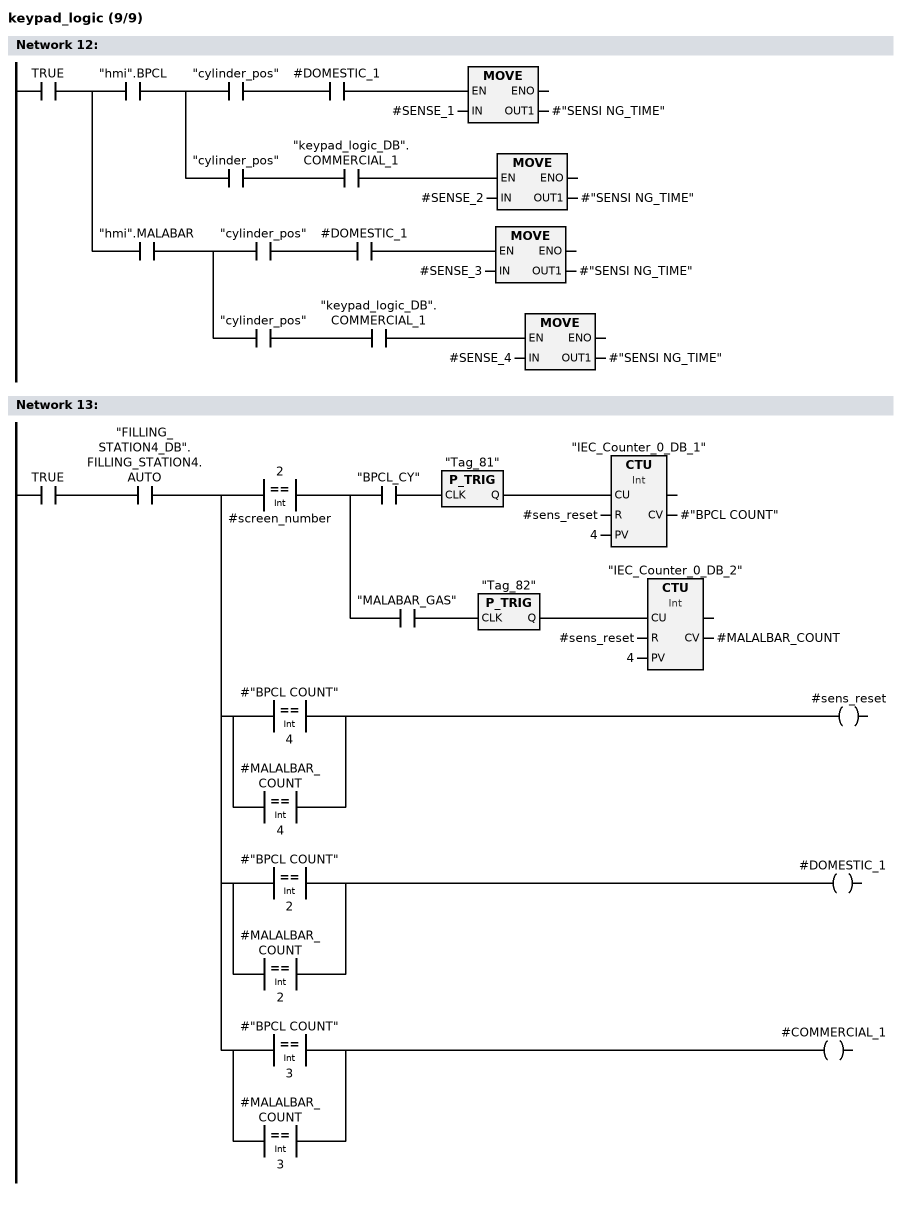
   RUNG wire#powerrail
      Contact( TRUE )
      wire#w1
      Contact( "hmi".BPCL )
      wire#w2
      Contact( "cylinder_pos" )
      Contact( #DOMESTIC_1 )
      Move(in := #SENSE_1, out1 => #"SENSI NG_TIME")
   END_RUNG
   RUNG wire#w2
      Contact( "cylinder_pos" )
      Contact( "keypad_logic_DB".COMMERCIAL_1 )
      Move(in := #SENSE_2, out1 => #"SENSI NG_TIME")
   END_RUNG
   RUNG wire#w1
      Contact( "hmi".MALABAR )
      wire#w3
      Contact( "cylinder_pos" )
      Contact( #DOMESTIC_1 )
      Move(in := #SENSE_3, out1 => #"SENSI NG_TIME")
   END_RUNG
   RUNG wire#w3
      Contact( "cylinder_pos" )
      Contact( "keypad_logic_DB".COMMERCIAL_1 )
      Move(in := #SENSE_4, out1 => #"SENSI NG_TIME")
   END_RUNG
   // the same network as SCL:
   #_w1 := TRUE AND "hmi".BPCL;
   IF #_w1 AND "cylinder_pos" AND #DOMESTIC_1 THEN #"SENSI NG_TIME" := #SENSE_1; END_IF;
   IF #_w1 AND "cylinder_pos" AND "keypad_logic_DB".COMMERCIAL_1 THEN #"SENSI NG_TIME" := #SENSE_2; END_IF;
   #_w2 := TRUE AND "hmi".MALABAR;
   IF #_w2 AND "cylinder_pos" AND #DOMESTIC_1 THEN #"SENSI NG_TIME" := #SENSE_3; END_IF;
   IF #_w2 AND "cylinder_pos" AND "keypad_logic_DB".COMMERCIAL_1 THEN #"SENSI NG_TIME" := #SENSE_4; END_IF;
END_REGION

REGION Network 13
   RUNG wire#powerrail
      Contact( TRUE )
      Contact( "FILLING_STATION4_DB".FILLING_STATION4.AUTO )
      wire#w1
      { S7_Templates := "SrcType := Int" } EQ_Contact(in1 := 2, in2 := #screen_number)
      wire#w2
      Contact( "BPCL_CY" )
      P_Trig( "Tag_81" )
      { S7_Templates := "value_type := Int" } "IEC_Counter_0_DB_1".CTU(r := #sens_reset, pv := 4, cv => #"BPCL COUNT")
   END_RUNG
   RUNG wire#w2
      Contact( "MALABAR_GAS" )
      P_Trig( "Tag_82" )
      { S7_Templates := "value_type := Int" } "IEC_Counter_0_DB_2".CTU(r := #sens_reset, pv := 4, cv => #MALALBAR_COUNT)
   END_RUNG
   RUNG wire#w1
      { S7_Templates := "SrcType := Int" } EQ_Contact(in1 := #"BPCL COUNT", in2 := 4)
      wire#w3
      Coil( #sens_reset )
   END_RUNG
   RUNG wire#w1
      { S7_Templates := "SrcType := Int" } EQ_Contact(in1 := #MALALBAR_COUNT, in2 := 4)
   END_RUNG wire#w3
   RUNG wire#w1
      { S7_Templates := "SrcType := Int" } EQ_Contact(in1 := #"BPCL COUNT", in2 := 2)
      wire#w4
      Coil( #DOMESTIC_1 )
   END_RUNG
   RUNG wire#w1
      { S7_Templates := "SrcType := Int" } EQ_Contact(in1 := #MALALBAR_COUNT, in2 := 2)
   END_RUNG wire#w4
   RUNG wire#w1
      { S7_Templates := "SrcType := Int" } EQ_Contact(in1 := #"BPCL COUNT", in2 := 3)
      wire#w5
      Coil( #COMMERCIAL_1 )
   END_RUNG
   RUNG wire#w1
      { S7_Templates := "SrcType := Int" } EQ_Contact(in1 := #MALALBAR_COUNT, in2 := 3)
   END_RUNG wire#w5
   // the same network as SCL:
   #_w1 := TRUE AND "FILLING_STATION4_DB".FILLING_STATION4.AUTO;
   #_w2 := #_w1 AND (2 = #screen_number);
   #_w3 := #_w2 AND "BPCL_CY";
   #_w4 := #_w3 AND NOT "Tag_81";   // rising edge
   "Tag_81" := #_w3;
   "IEC_Counter_0_DB_1".CTU(CU := #_w4, R := #sens_reset, PV := 4, CV => #"BPCL COUNT");
   #_w5 := #_w2 AND "MALABAR_GAS";
   #_w6 := #_w5 AND NOT "Tag_82";   // rising edge
   "Tag_82" := #_w5;
   "IEC_Counter_0_DB_2".CTU(CU := #_w6, R := #sens_reset, PV := 4, CV => #MALALBAR_COUNT);
   #sens_reset := #_w1 AND ((#"BPCL COUNT" = 4) OR (#MALALBAR_COUNT = 4));
   #DOMESTIC_1 := #_w1 AND ((#"BPCL COUNT" = 2) OR (#MALALBAR_COUNT = 2));
   #COMMERCIAL_1 := #_w1 AND ((#"BPCL COUNT" = 3) OR (#MALALBAR_COUNT = 3));
END_REGION
END_FUNCTION_BLOCK
